{attribute 'qualified_only'}
VAR_GLOBAL
	
	aCameraConfig	: ARRAY[1..2] OF ST_SCANNER_Configuration;
	aCameraStatus	: ARRAY[1..2] OF ST_SCANNER_Status;
	aCameraControl	: ARRAY[1..2] OF ST_SCANNER_Ctrl;
END_VAR

(* stored: Version 1.1.0.1
   GVL gCamDevice: Id {0a9de249-9e7c-4f5f-9a59-8c263128b5ba} *)
